FUNCTION_BLOCK FB_012_StepOnAfterStopEx

VAR_INPUT
	bExecute:BOOL;
END_VAR
VAR_OUTPUT
	bBusy:BOOL;(*功能块执行忙标志*)
	bError:BOOL;(*出错*)
	bDone:BOOL;(*执行完毕*)
END_VAR
VAR_IN_OUT
//	stX:AXIS_REF;
//	stY:AXIS_REF;
//	stZ:AXIS_REF;
	stItpToPlc :NCTOPLC_NCICHANNEL_REF;
	stPlcToItp:PLCTONC_NCICHANNEL_REF;
END_VAR
VAR
	AfterStopStep:INT:=0;
	fbsteponafterestop:ItpStepOnAfterEStopEx;(*暂停重启*)
END_VAR

CASE AfterStopStep OF
	0:
	  IF  bExecute THEN
		 bBusy:=TRUE;(*FB执行状态*)
		 bDone:=FALSE;(*FB执行完毕*)
		 bError:=FALSE;(*报错*)
		 AfterStopStep:=10;(*进入10步*) 
	  END_IF
	10:
	  fbsteponafterestop(
	    bExecute:= TRUE, 
	    tTimeOut:= , 
	    sNciToPlc:= stItpToPlc, 
	    bBusy=> , 
	    bErr=> , 
	    nErrId=> );
	   IF NOT fbsteponafterestop.bBusy THEN
		  IF NOT fbsteponafterestop.bErr THEN
			AfterStopStep:=20;(*进入20步*)  
		  ELSE
			bBusy:=FALSE;
			bError:=TRUE;
			AfterStopStep:=999;
		  END_IF
		  fbsteponafterestop(bExecute:= FALSE,sNciToPlc:= stItpToPlc); 
	    END_IF
	 20:
	   bDone:=TRUE;
       bBusy:=FALSE;   
	   IF NOT bExecute THEN
		 AfterStopStep:=0;
	   END_IF
	 999:
	   IF NOT bExecute THEN		   
	    AfterStopStep:=0;
        bError:=FALSE; 
	   END_IF
END_CASE

END_FUNCTION_BLOCK

(* stored: Version 1.1.0.1, ProductVersion 3.1.4024.12
   POU FB_012_StepOnAfterStopEx: Id {2001fb99-efae-41a1-acb9-572981cb56a8}, SpecialFunc None *)
